// Mitsubishi GX Works2 project: ZP_funtion   PLC: Q03UDV

PROGRAM MAIN
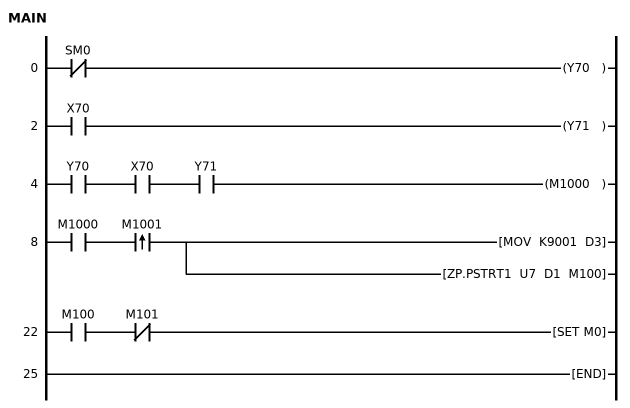
0     LDI     SM0
      OUT     Y70
2     LD      X70
      OUT     Y71
4     LD      Y70
      AND     X70
      AND     Y71
      OUT     M1000
8     LD      M1000
      ANDP    M1001
      MOV     K9001 D3
      ZP.PSTRT1 U7 D1 M100
22    LD      M100
      ANI     M101
      SET     M0
25    END
END_PROGRAM
